Fanuc TP program (LS listing): B002003.LS

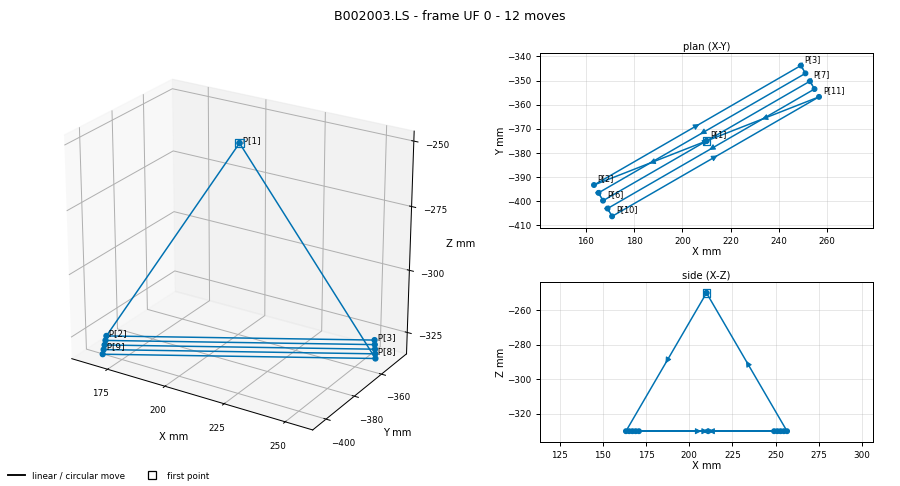
[picture p0: tool path of B002003.LS in frame UF 0, 12 of 12 moves have a stored position in this frame; points joined in program order, loops and branches not executed]
/PROG  B002003.LS
/ATTR
OWNER       = MNEDITOR;
COMMENT     = "";
PROG_SIZE   = 636;
CREATE      = DATE 23-01-07  TIME 11:59:14;
MODIFIED    = DATE 23-01-07  TIME 12:02:18;
FILE_NAME   = ;
VERSION     = 0;
LINE_COUNT  = 4;
MEMORY_SIZE = 992;
PROTECT     = READ_WRITE;
TCD:  STACK_SIZE	= 0,
      TASK_PRIORITY	= 50,
      TIME_SLICE	= 0,
      BUSY_LAMP_OFF	= 0,
      ABORT_REQUEST	= 0,
      PAUSE_REQUEST	= 0;
DEFAULT_GROUP	= 1,*,*,*,*;
CONTROL_CODE	= 00000000 00000000;
/MN
   1:J P[1] 100% FINE    ;
   2:L P[2] 100mm/sec CNT100    ;
   3:L P[3] 100mm/sec CNT100    ;
   4:L P[4] 100mm/sec CNT100    ;
   5:L P[5] 100mm/sec CNT100    ;
   6:L P[6] 100mm/sec CNT100    ;
   7:L P[7] 100mm/sec CNT100    ;
   8:L P[8] 100mm/sec CNT100    ;
   9:L P[9] 100mm/sec CNT100    ;
   10:L P[10] 100mm/sec CNT100    ;
   11:L P[11] 100mm/sec CNT100    ;
   12:L P[12] 100mm/sec CNT100    ;
/POS
P[1]{
   GP1:
	UF : 0, UT : 6,		CONFIG : 'N U T, 0, 0, 0',
	X =  210.000  mm,	Y =   -375.000  mm,	Z =   -250.000  mm,
	W =  90.000 deg,	P =   0.000 deg,	R =   90.000 deg
};
P[2]{
   GP1:
	UF : 0, UT : 6,		CONFIG : 'N U T, 0, 0, 0',
	X =  163.392  mm,	Y =   -393.255  mm,	Z =   -330.000  mm,
	W =  90.000 deg,	P =   0.000 deg,	R =   90.000 deg
};
P[3]{
   GP1:
	UF : 0, UT : 6,		CONFIG : 'N U T, 0, 0, 0',
	X =  249.114  mm,	Y =   -343.760  mm,	Z =   -330.000  mm,
	W =  90.000 deg,	P =   0.000 deg,	R =   90.000 deg
};
P[4]{
   GP1:
	UF : 0, UT : 6,		CONFIG : 'N U T, 0, 0, 0',
	X =  250.988  mm,	Y =   -347.006  mm,	Z =   -330.000  mm,
	W =  90.000 deg,	P =   0.000 deg,	R =   90.000 deg
};
P[5]{
   GP1:
	UF : 0, UT : 6,		CONFIG : 'N U T, 0, 0, 0',
	X =  165.266  mm,	Y =   -396.501  mm,	Z =   -330.000  mm,
	W =  90.000 deg,	P =   0.000 deg,	R =   90.000 deg
};
P[6]{
   GP1:
	UF : 0, UT : 6,		CONFIG : 'N U T, 0, 0, 0',
	X =  167.140  mm,	Y =   -399.747  mm,	Z =   -330.000  mm,
	W =  90.000 deg,	P =   0.000 deg,	R =   90.000 deg
};
P[7]{
   GP1:
	UF : 0, UT : 6,		CONFIG : 'N U T, 0, 0, 0',
	X =  252.862  mm,	Y =   -350.252  mm,	Z =   -330.000  mm,
	W =  90.000 deg,	P =   0.000 deg,	R =   90.000 deg
};
P[8]{
   GP1:
	UF : 0, UT : 6,		CONFIG : 'N U T, 0, 0, 0',
	X =  254.736  mm,	Y =   -353.498  mm,	Z =   -330.000  mm,
	W =  90.000 deg,	P =   0.000 deg,	R =   90.000 deg
};
P[9]{
   GP1:
	UF : 0, UT : 6,		CONFIG : 'N U T, 0, 0, 0',
	X =  169.014  mm,	Y =   -402.993  mm,	Z =   -330.000  mm,
	W =  90.000 deg,	P =   0.000 deg,	R =   90.000 deg
};
P[10]{
   GP1:
	UF : 0, UT : 6,		CONFIG : 'N U T, 0, 0, 0',
	X =  170.889  mm,	Y =   -406.238  mm,	Z =   -330.000  mm,
	W =  90.000 deg,	P =   0.000 deg,	R =   90.000 deg
};
P[11]{
   GP1:
	UF : 0, UT : 6,		CONFIG : 'N U T, 0, 0, 0',
	X =  256.610  mm,	Y =   -356.744  mm,	Z =   -330.000  mm,
	W =  90.000 deg,	P =   0.000 deg,	R =   90.000 deg
};
P[12]{
   GP1:
	UF : 0, UT : 6,		CONFIG : 'N U T, 0, 0, 0',
	X =  210.000  mm,	Y =   -375.000  mm,	Z =   -250.000  mm,
	W =  90.000 deg,	P =   0.000 deg,	R =   90.000 deg
};
/END
